FUNCTION normProjIdx : DINT
VAR_INPUT
	idx: DINT;
	size: DINT;
END_VAR
VAR
	tmp: DINT;
END_VAR

tmp := idx;
IF tmp < 0 THEN
    tmp := size + tmp;
END_IF;
normProjIdx := tmp;

END_FUNCTION

(* stored: Version 1.1.0.1, ProductVersion 3.1.4022.18
   POU normProjIdx: Id {ad98ab73-384a-4b76-a461-fc8a4b6dfa59}, SpecialFunc None *)
